TYPE ST_SAFETY_FBCONNECTIONSHUTDOWN:
STRUCT
	uStatus							: U_SAFETY_CONNECTIONSHUTDOWN; 		(* Typ zalezny od bloku *)
	eState							: E_SAFETY_FBStateCS;				(* Enum ze statusem bloku *)
	bGeneralError					: BOOL; 							(* Gdy wystapi chociaz jeden Error *)	
END_STRUCT
END_TYPE

(* stored: Version 1.1.0.1, ProductVersion 3.1.4022.12
   DUT ST_SAFETY_FBCONNECTIONSHUTDOWN: Id {b29e70d1-e765-4c2a-b01e-fff332d3b9cb} *)
